// Mitsubishi GX Works2 project: PLC1_E2   PLC: FX3G

// global labels: Global1
VAR_GLOBAL
  dayStart AT X007 : BOOL;
  workday AT Y007 : BOOL;
  Emergency AT X005 : BOOL;
  chocolate AT CS0 : BOOL;
  nuts AT CS1 : BOOL;
  pistachio AT CS2 : BOOL;
  kadayif AT CS3 : BOOL;
  choco AT CC0 : BOOL;
  nut AT CC1 : BOOL;
  pistachi AT CC2 : BOOL;
  kadayifi AT CC3 : BOOL;
  analog_output AT D8282 : INT;
END_VAR
VAR_GLOBAL CONSTANT
  chocolate_input : REAL := 1200;
END_VAR
VAR_GLOBAL
  chocolate_inventory AT D1120 : REAL;
END_VAR
VAR_GLOBAL CONSTANT
  nuts_input : REAL := 300;
  choolate_inventory : REAL := 300;
END_VAR
VAR_GLOBAL
  nuts_inventory AT D1130 : REAL;
END_VAR
VAR_GLOBAL CONSTANT
  pistachio_input : REAL := 300;
END_VAR
VAR_GLOBAL
  pistachio_inventory AT D1140 : REAL;
END_VAR
VAR_GLOBAL CONSTANT
  kadayif_input : REAL := 120;
END_VAR
VAR_GLOBAL
  kadayif_inventory AT D1150 : REAL;
  gotChocolate AT M10 : BOOL;
END_VAR
VAR_GLOBAL CONSTANT
  chocolateMinReq : REAL := 400.0;
END_VAR
VAR_GLOBAL
  gotNuts AT M11 : BOOL;
END_VAR
VAR_GLOBAL CONSTANT
  nutsMinReq : REAL := 100.0;
END_VAR
VAR_GLOBAL
  gotPistachio AT M12 : BOOL;
END_VAR
VAR_GLOBAL CONSTANT
  PistachioMinReq : REAL := 120.0;
END_VAR
VAR_GLOBAL
  gotKadayif AT M13 : BOOL;
END_VAR
VAR_GLOBAL CONSTANT
  KadayifMinReq : REAL := 60.0;
END_VAR
VAR_GLOBAL
  possibleManufacture AT M1 : BOOL;
  startMelting AT X001 : BOOL;
END_VAR
VAR_GLOBAL CONSTANT
  chocolateAmount : REAL := 400;
END_VAR
VAR_GLOBAL
  timerFinished AT TS1 : BOOL;
  meltInProgress AT Y001 : BOOL;
  meltIngTimer AT TC1 : BOOL;
  heatSensor AT X002 : BOOL;
  startCasting AT X003 : BOOL;
  castInProgress AT Y002 : BOOL;
  castingTimer AT TC1 : BOOL;
END_VAR
VAR_GLOBAL CONSTANT
  constantCastingTime : INT := 40;
END_VAR
VAR_GLOBAL
  startFilling AT X004 : BOOL;
  analog_input AT D8280 : INT;
  analog_input_div AT D170 : REAL;
END_VAR
VAR_GLOBAL CONSTANT
  nutsMixConstant : REAL := 5;
END_VAR
VAR_GLOBAL
  nutsMix AT M2 : BOOL;
END_VAR
VAR_GLOBAL CONSTANT
  dubaiConstant : REAL := 5.0;
END_VAR
VAR_GLOBAL
  dubai AT M3 : BOOL;
  sensorStartCasting AT X003 : BOOL;
END_VAR
VAR_GLOBAL CONSTANT
  dubaiConstantUpper : INT := 10;
  ratio : REAL := 400;
  nutsForNutsMix : REAL := 100;
  pistachioForNutsMix : REAL := 100;
  nutsForDubai : REAL := 20;
  pistachioForDubai : REAL := 120;
  kadayifForDubai : REAL := 60;
END_VAR
VAR_GLOBAL
  fillingTimer AT TC2 : BOOL;
END_VAR
VAR_GLOBAL CONSTANT
  fillingTime_5sec : INT := 50;
END_VAR
VAR_GLOBAL
  finishFilling AT TS2 : BOOL;
  flashingRound AT M5 : BOOL;
  bulb3Timer AT TC3 : BOOL;
END_VAR
VAR_GLOBAL CONSTANT
  flashingConstant : INT := 5;
END_VAR
VAR_GLOBAL
  bulb3Finish AT TS3 : BOOL;
  bulb3 AT Y003 : BOOL;
  bulb4Timer AT TC4 : BOOL;
  bulb4Finish AT TS4 : BOOL;
  bulb4 AT Y004 : BOOL;
  startCooling AT X006 : BOOL;
  coolingTimer AT TC5 : BOOL;
  coolingInProgress AT Y006 : BOOL;
  coolingFinished AT TS5 : BOOL;
END_VAR
VAR_GLOBAL CONSTANT
  constantCoolingTime : INT := 30;
END_VAR
VAR_GLOBAL
  tables_in_package_counter AT CC4 : BOOL;
  startPacking AT X000 : BOOL;
END_VAR
VAR_GLOBAL CONSTANT
  tablesInPack_4 : INT := 4;
END_VAR
VAR_GLOBAL
  four_tables_packed AT CS4 : BOOL;
  current_tables_packed AT CN4 : INT;
END_VAR
VAR_GLOBAL CONSTANT
  const_1 : INT := 1;
  const_5 : INT := 5;
END_VAR
VAR_GLOBAL
  packingBulb AT Y005 : BOOL;
  cooling_finished AT TS5 : BOOL;
  cooling_indicator AT M20 : BOOL;
END_VAR
VAR_GLOBAL CONSTANT
  const_4 : INT := 4;
  const_3 : INT := 3;
END_VAR
VAR_GLOBAL
  pack_num AT D1160 : INT;
  TEST AT X011 : BOOL;
  TESTING AT Y011 : BOOL;
  TESRRR AT Y002 : BOOL;
  HELP AT X011 : BOOL;
END_VAR
VAR_GLOBAL CONSTANT
  constantCastTime : INT := 40;
END_VAR
VAR_GLOBAL
  analog_real1 AT D1200 : REAL;
  finish_input_analog1 AT M21 : BOOL;
  melt_complete AT M30 : BOOL;
  nutsMix_finish AT M32 : BOOL;
  dubai_finish AT M33 : BOOL;
  finish_casting AT M30 : BOOL;
  packingInProgress AT M40 : BOOL;
  filling_chosen AT M34 : BOOL;
  input_chosen AT M39 : BOOL;
END_VAR
VAR_GLOBAL CONSTANT
  const_0_1 : REAL := 0.1;
END_VAR
VAR_GLOBAL
  switchesOff AT M40 : BOOL;
  castingFinished AT M4 : BOOL;
  output_storage AT D1160 : REAL;
END_VAR
VAR_GLOBAL CONSTANT
  const40 : REAL := 40;
  const20 : REAL := 20;
END_VAR
VAR_GLOBAL
  newIteration AT M6 : BOOL;
  iterationGoing AT M7 : BOOL;
END_VAR
VAR_GLOBAL CONSTANT
  const400 : REAL := 400;
  const1 : REAL := 1.0;
END_VAR

// task Task_01 (event TRUE, interval 0, priority 31): POU_01

PROGRAM POU_01
(* structured ladder/FBD written out as ST: instructions are called as NAME(EN, inputs, outputs); _pN, _eN, _tN stand for wires *)
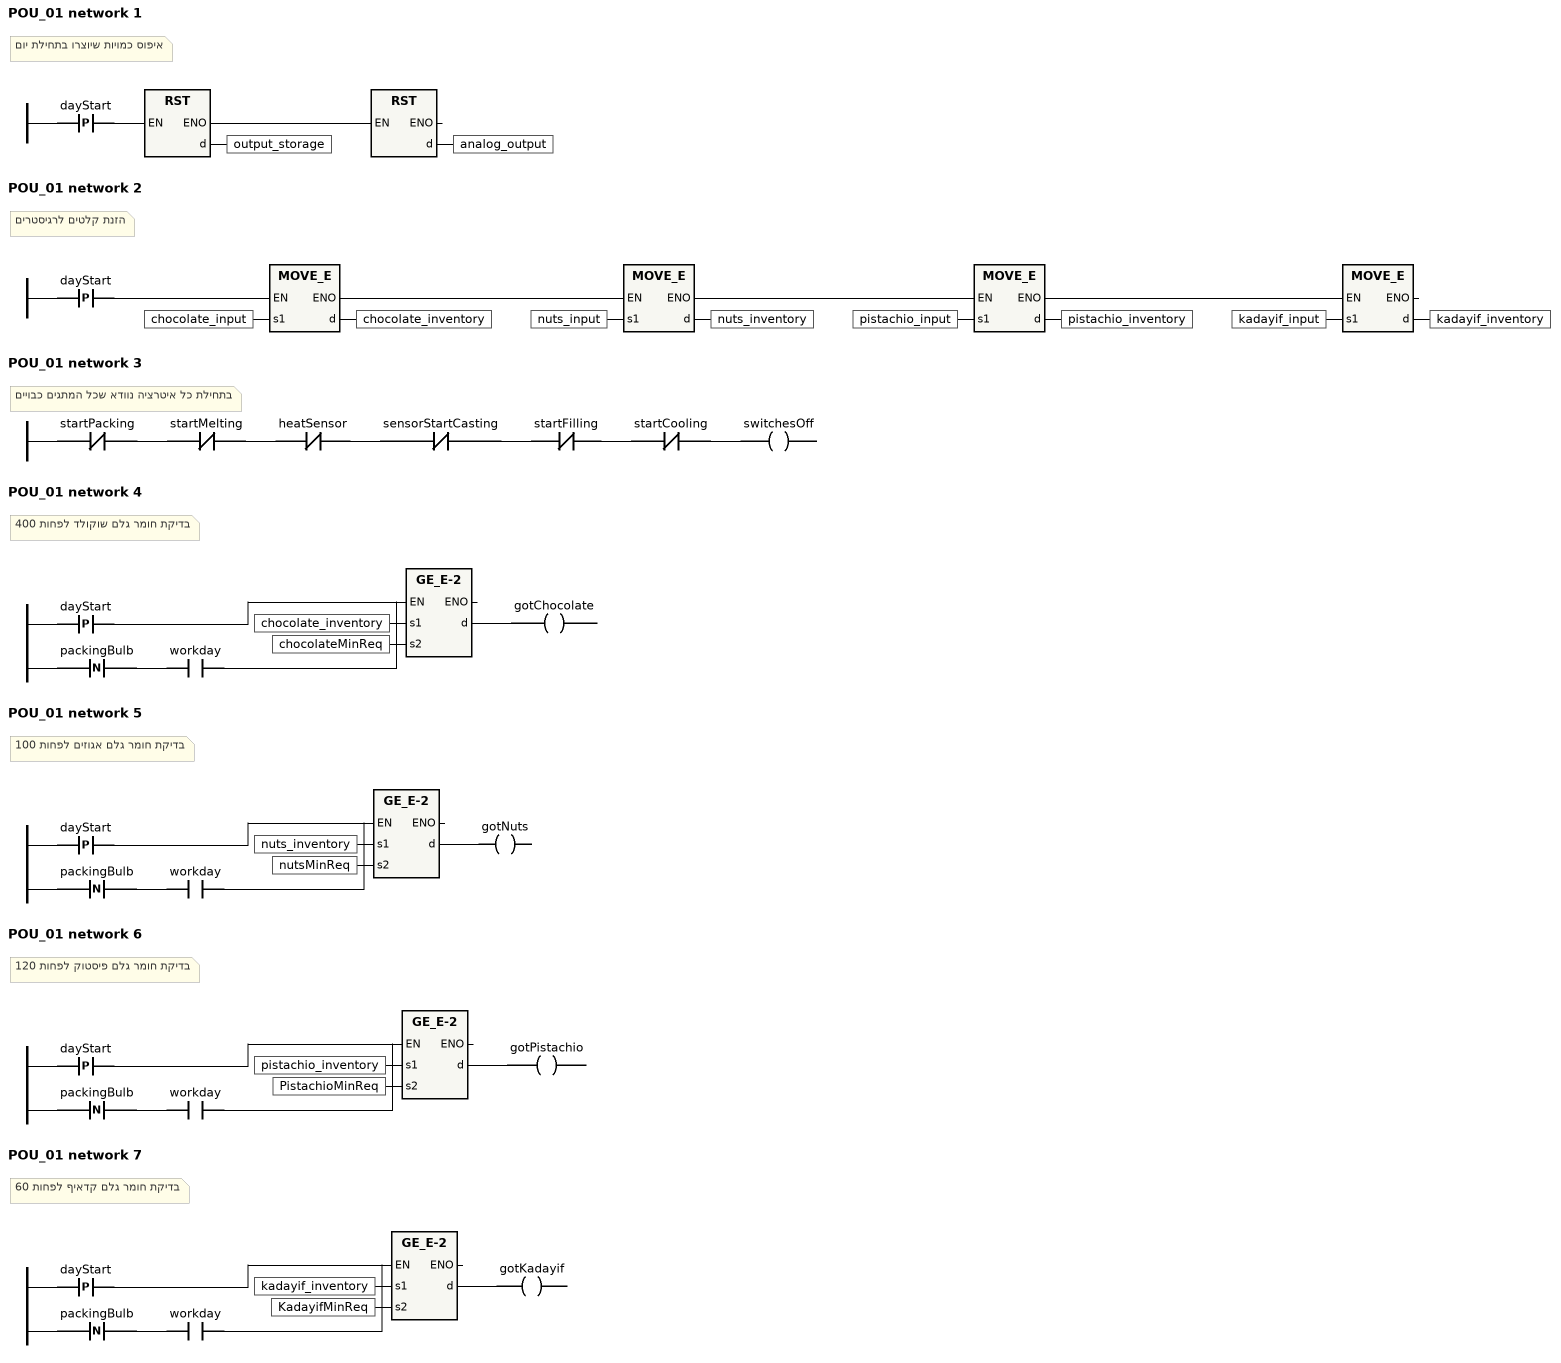
(* network 1 *)
(* איפוס כמויות שיוצרו בתחילת יום *)
_e1 := RST(LDP(TRUE, dayStart), output_storage);
RST(_e1, analog_output);
(* network 2 *)
(* הזנת קלטים לרגיסטרים *)
_e1 := MOVE_E(LDP(TRUE, dayStart), chocolate_input, chocolate_inventory);
_e2 := MOVE_E(_e1, nuts_input, nuts_inventory);
_e3 := MOVE_E(_e2, pistachio_input, pistachio_inventory);
MOVE_E(_e3, kadayif_input, kadayif_inventory);
(* network 3 *)
(* בתחילת כל איטרציה נוודא שכל המתגים כבויים *)
switchesOff := NOT startPacking AND NOT startMelting AND NOT heatSensor AND NOT sensorStartCasting AND NOT startFilling AND NOT startCooling;
(* network 4 *)
(* בדיקת חומר גלם שוקולד לפחות 400 *)
GE_E(LDP(TRUE, dayStart) OR (LDF(TRUE, packingBulb) AND workday), chocolate_inventory, chocolateMinReq, _t1);
gotChocolate := _t1;
(* network 5 *)
(* בדיקת חומר גלם אגוזים לפחות 100 *)
GE_E(LDP(TRUE, dayStart) OR (LDF(TRUE, packingBulb) AND workday), nuts_inventory, nutsMinReq, _t1);
gotNuts := _t1;
(* network 6 *)
(* בדיקת חומר גלם פיסטוק לפחות 120 *)
GE_E(LDP(TRUE, dayStart) OR (LDF(TRUE, packingBulb) AND workday), pistachio_inventory, PistachioMinReq, _t1);
gotPistachio := _t1;
(* network 7 *)
(* בדיקת חומר גלם קדאיף לפחות 60 *)
GE_E(LDP(TRUE, dayStart) OR (LDF(TRUE, packingBulb) AND workday), kadayif_inventory, KadayifMinReq, _t1);
gotKadayif := _t1;
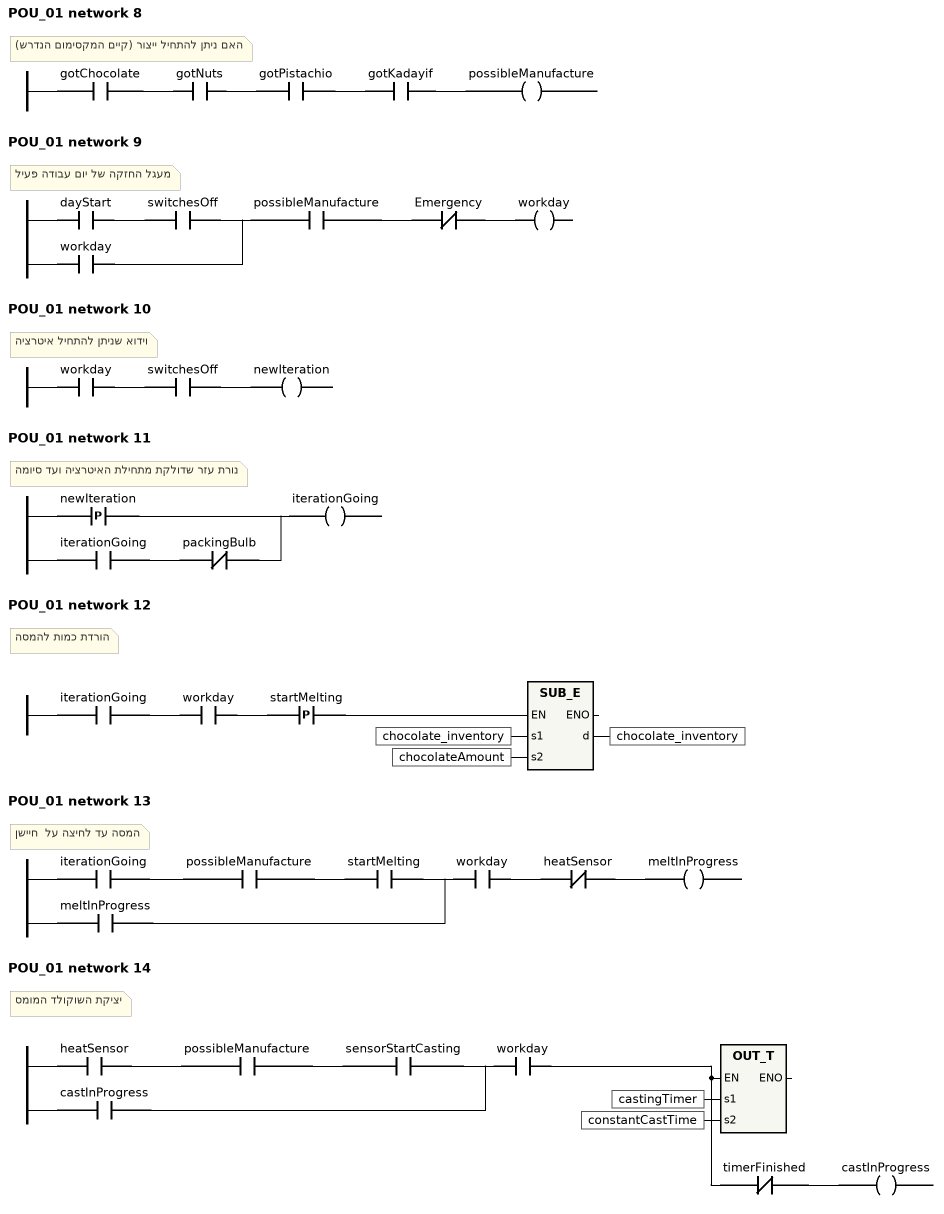
(* network 8 *)
(* האם ניתן להתחיל ייצור (קיים המקסימום הנדרש) *)
possibleManufacture := gotChocolate AND gotNuts AND gotPistachio AND gotKadayif;
(* network 9 *)
(* מעגל החזקה של יום עבודה פעיל *)
workday := (((dayStart AND switchesOff) OR workday) AND possibleManufacture) AND NOT Emergency;
(* network 10 *)
(* וידוא שניתן להתחיל איטרציה *)
newIteration := workday AND switchesOff;
(* network 11 *)
(* נורת עזר שדולקת מתחילת האיטרציה ועד סיומה *)
iterationGoing := LDP(TRUE, newIteration) OR (iterationGoing AND NOT packingBulb);
(* network 12 *)
(* הורדת כמות להמסה *)
SUB_E(iterationGoing AND workday AND LDP(TRUE, startMelting), chocolate_inventory, chocolateAmount, chocolate_inventory);
(* network 13 *)
(* המסה עד לחיצה על  חיישן *)
meltInProgress := (((iterationGoing AND possibleManufacture AND startMelting) OR meltInProgress) AND workday) AND NOT heatSensor;
(* network 14 *)
(* יציקת השוקולד המומס *)
_p1 := ((heatSensor AND possibleManufacture AND sensorStartCasting) OR castInProgress) AND workday;
castInProgress := _p1 AND NOT timerFinished;
OUT_T(_p1, castingTimer, constantCastTime);
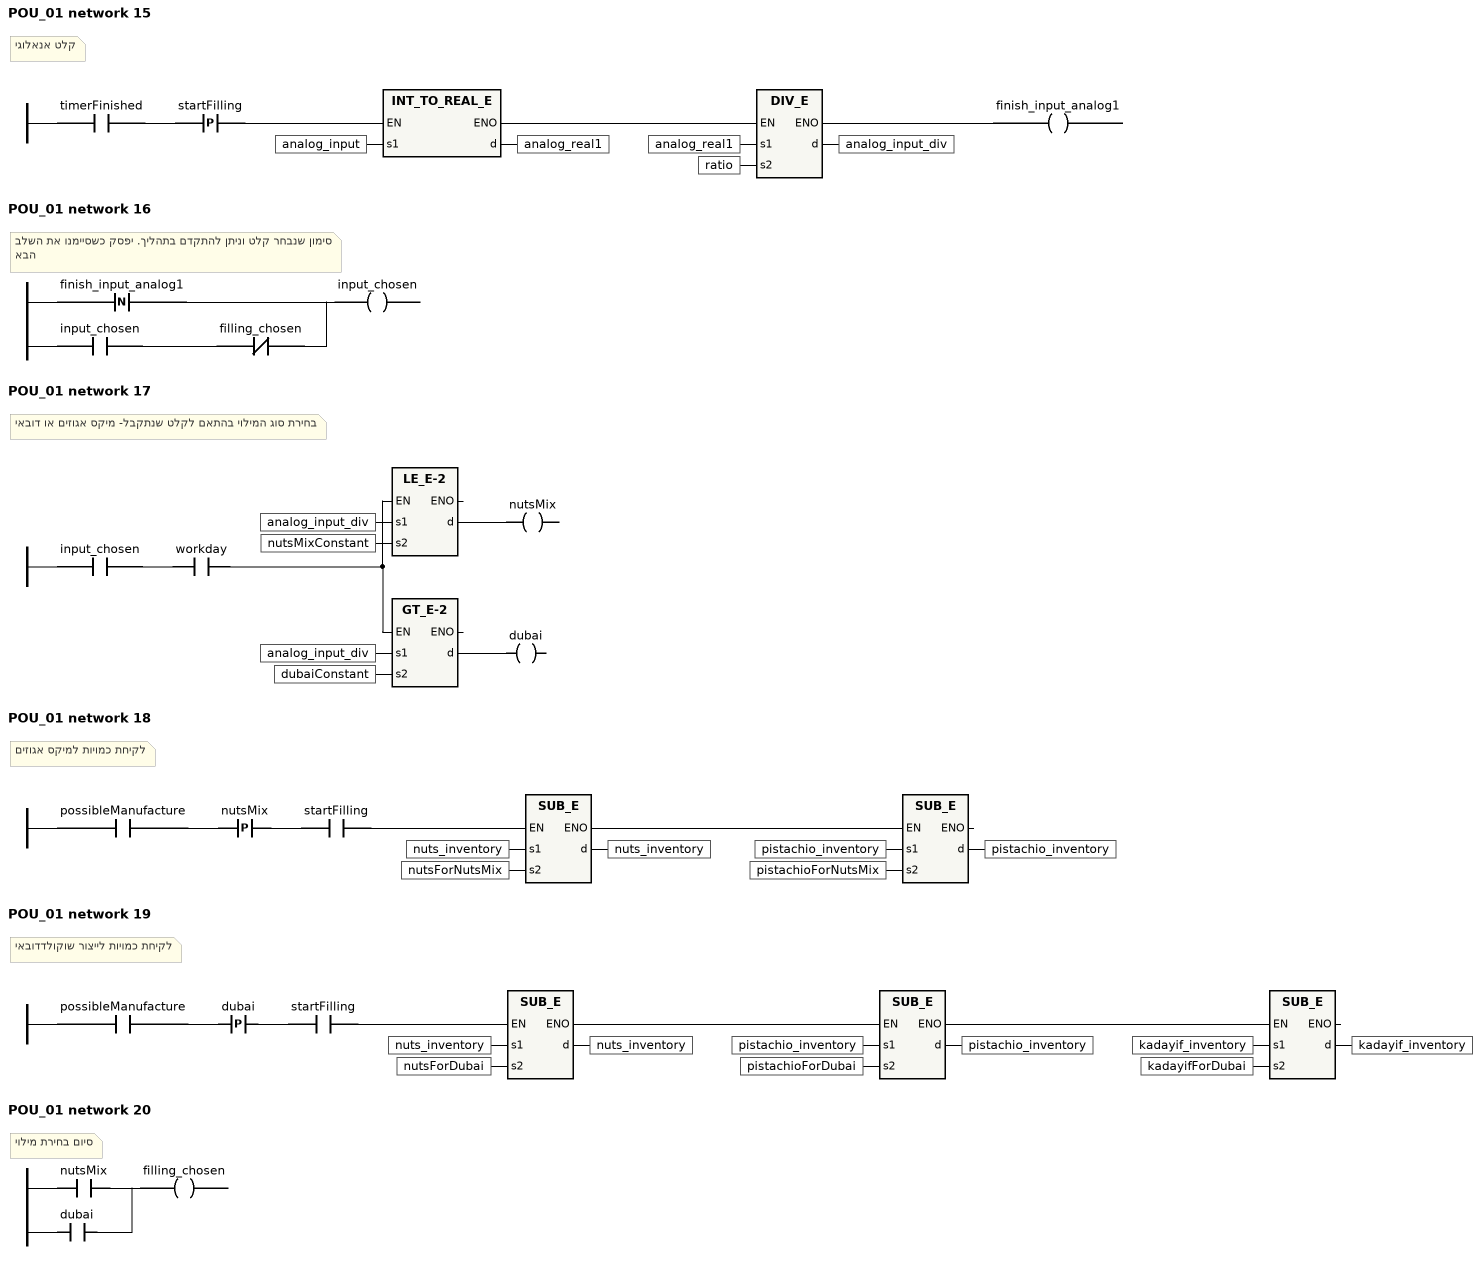
(* network 15 *)
(* קלט אנאלוגי *)
_e1 := INT_TO_REAL_E(timerFinished AND LDP(TRUE, startFilling), analog_input, analog_real1);
_e2 := DIV_E(_e1, analog_real1, ratio, analog_input_div);
finish_input_analog1 := _e2;
(* network 16 *)
(* סימון שנבחר קלט וניתן להתקדם בתהליך. יפסק כשסיימנו את השלב הבא *)
input_chosen := LDF(TRUE, finish_input_analog1) OR (input_chosen AND NOT filling_chosen);
(* network 17 *)
(* בחירת סוג המילוי בהתאם לקלט שנתקבל- מיקס אגוזים או דובאי *)
_p1 := input_chosen AND workday;
LE_E(_p1, analog_input_div, nutsMixConstant, _t2);
nutsMix := _t2;
GT_E(_p1, analog_input_div, dubaiConstant, _t3);
dubai := _t3;
(* network 18 *)
(* לקיחת כמויות למיקס אגוזים *)
_e1 := SUB_E(possibleManufacture AND LDP(TRUE, nutsMix) AND startFilling, nuts_inventory, nutsForNutsMix, nuts_inventory);
SUB_E(_e1, pistachio_inventory, pistachioForNutsMix, pistachio_inventory);
(* network 19 *)
(* לקיחת כמויות לייצור שוקולדדובאי *)
_e1 := SUB_E(possibleManufacture AND LDP(TRUE, dubai) AND startFilling, nuts_inventory, nutsForDubai, nuts_inventory);
_e2 := SUB_E(_e1, pistachio_inventory, pistachioForDubai, pistachio_inventory);
SUB_E(_e2, kadayif_inventory, kadayifForDubai, kadayif_inventory);
(* network 20 *)
(* סיום בחירת מילוי *)
filling_chosen := nutsMix OR dubai;
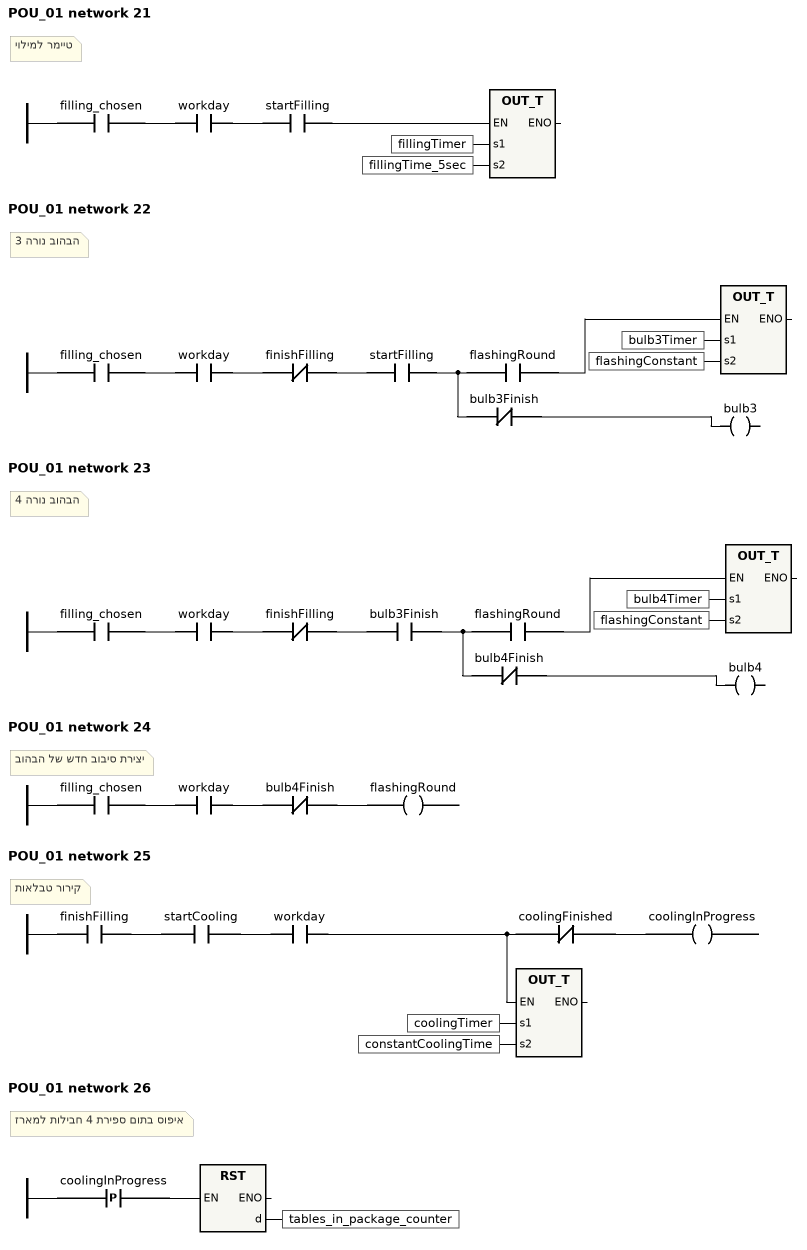
(* network 21 *)
(* טיימר למילוי *)
OUT_T(filling_chosen AND workday AND startFilling, fillingTimer, fillingTime_5sec);
(* network 22 *)
(* הבהוב נורה 3 *)
_p1 := filling_chosen AND workday AND NOT finishFilling AND startFilling;
OUT_T(_p1 AND flashingRound, bulb3Timer, flashingConstant);
bulb3 := _p1 AND NOT bulb3Finish;
(* network 23 *)
(* הבהוב נורה 4 *)
_p1 := filling_chosen AND workday AND NOT finishFilling AND bulb3Finish;
OUT_T(_p1 AND flashingRound, bulb4Timer, flashingConstant);
bulb4 := _p1 AND NOT bulb4Finish;
(* network 24 *)
(* יצירת סיבוב חדש של הבהוב *)
flashingRound := filling_chosen AND workday AND NOT bulb4Finish;
(* network 25 *)
(* קירור טבלאות *)
_p1 := finishFilling AND startCooling AND workday;
coolingInProgress := _p1 AND NOT coolingFinished;
OUT_T(_p1, coolingTimer, constantCoolingTime);
(* network 26 *)
(* איפוס בתום ספירת 4 חבילות למארז *)
RST(LDP(TRUE, coolingInProgress), tables_in_package_counter);
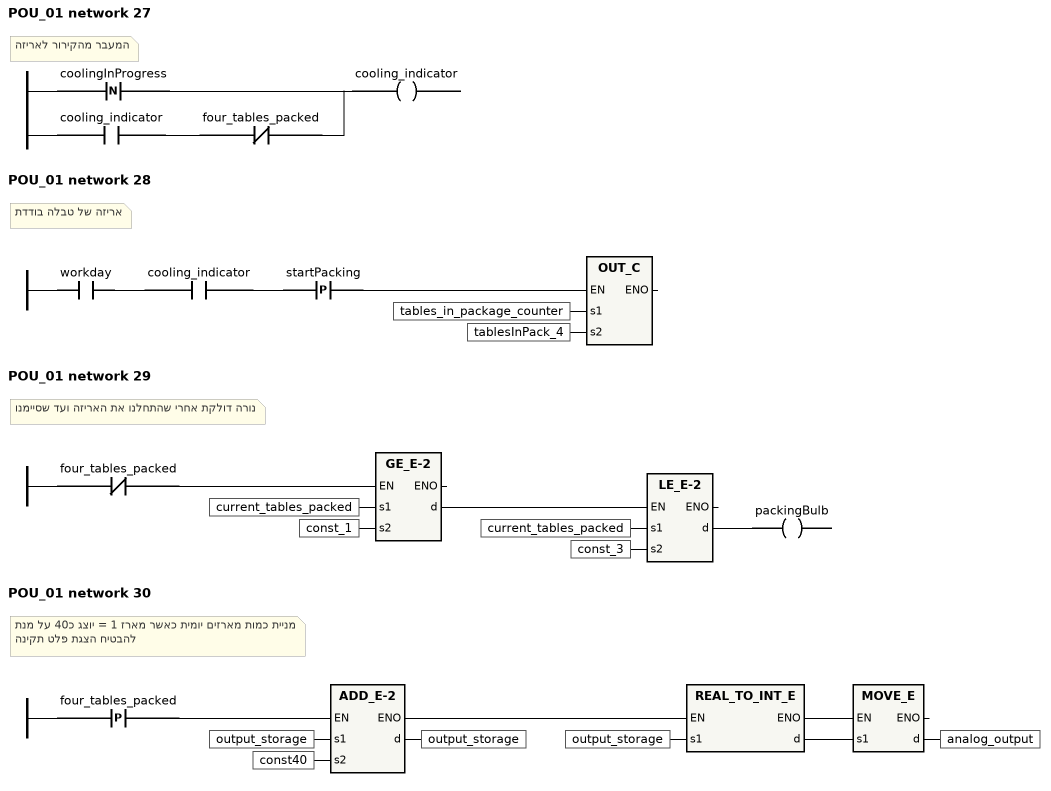
(* network 27 *)
(* המעבר מהקירור לאריזה *)
cooling_indicator := LDF(TRUE, coolingInProgress) OR (cooling_indicator AND NOT four_tables_packed);
(* network 28 *)
(* אריזה של טבלה בודדת *)
OUT_C(workday AND cooling_indicator AND LDP(TRUE, startPacking), tables_in_package_counter, tablesInPack_4);
(* network 29 *)
(* נורה דולקת אחרי שהתחלנו את האריזה ועד שסיימנו *)
GE_E(NOT four_tables_packed, current_tables_packed, const_1, _t1);
LE_E(_t1, current_tables_packed, const_3, _t2);
packingBulb := _t2;
(* network 30 *)
(* מניית כמות מארזים יומית כאשר מארז 1 = יוצג כ40 על מנת להבטיח הצגת פלט תקינה *)
_e1 := ADD_E(LDP(TRUE, four_tables_packed), output_storage, const40, output_storage);
_e3 := REAL_TO_INT_E(_e1, output_storage, _t2);
MOVE_E(_e3, _t2, analog_output);
END_PROGRAM
